// TIA Portal V20 export
TYPE "LER_typeServoTorqueCalControlNode"
// stored: Access Published
   STRUCT
      commands : "LER_typeServoTorqueCalCommands";
      monitoring : "LER_typeServoTorqueCalMonitoring";
   END_STRUCT;
END_TYPE
